PROGRAM prgCS4
VAR
	fbAlfen1					: FB_ECS_Alfen_NG9xx_Platform;						//{#lynus.ag#()}
	fbAlfen2					: FB_ECS_Alfen_NG9xx_Platform;						//{#lynus.ag#()}
	fbAlfen3					: FB_ECS_Alfen_NG9xx_Platform;						//{#lynus.ag#()}
	fbAlfen4					: FB_ECS_Alfen_NG9xx_Platform;						//{#lynus.ag#()}
	fbAlfen5					: FB_ECS_Alfen_NG9xx_Platform;						//{#lynus.ag#()}
	fbAlfen6					: FB_ECS_Alfen_NG9xx_Platform;						//{#lynus.ag#()}
	fbAlfen7					: FB_ECS_Alfen_NG9xx_Platform;						//{#lynus.ag#()}
	fbAlfen8					: FB_ECS_Alfen_NG9xx_Platform;						//{#lynus.ag#()}
	fbAlfen9					: FB_ECS_Alfen_NG9xx_Platform;						//{#lynus.ag#()}
	fbAlfen10					: FB_ECS_Alfen_NG9xx_Platform;						//{#lynus.ag#()}
	
	byErrorWarningUV1_1			: BYTE;												//{#lynus.ag#()}
	rChargingTimeInMinUV1_1		: REAL;												//{#lynus.ag#()}
	lrPowerUV1_1				: LREAL;											//{#lynus.ag#()}
	wStateUV1_1					: WORD;												//{#lynus.ag#()}
	lrEnergySessionUV1_1		: LREAL;											//{#lynus.ag#()}
	lrTotalEnergyUV1_1			: LREAL;											//{#lynus.ag#()}
	
	byErrorWarningUV1_2			: BYTE;												//{#lynus.ag#()}
	rChargingTimeInMinUV1_2		: REAL;												//{#lynus.ag#()}
	lrPowerUV1_2				: LREAL;											//{#lynus.ag#()}
	wStateUV1_2					: WORD;												//{#lynus.ag#()}
	lrEnergySessionUV1_2		: LREAL;											//{#lynus.ag#()}
	lrTotalEnergyUV1_2			: LREAL;											//{#lynus.ag#()}
	
	byErrorWarningUV1_3			: BYTE;												//{#lynus.ag#()}
	rChargingTimeInMinUV1_3		: REAL;												//{#lynus.ag#()}
	lrPowerUV1_3				: LREAL;											//{#lynus.ag#()}
	wStateUV1_3					: WORD;												//{#lynus.ag#()}
	lrEnergySessionUV1_3		: LREAL;											//{#lynus.ag#()}
	lrTotalEnergyUV1_3			: LREAL;											//{#lynus.ag#()}
	
	byErrorWarningUV1_4			: BYTE;												//{#lynus.ag#()}
	rChargingTimeInMinUV1_4		: REAL;												//{#lynus.ag#()}
	lrPowerUV1_4				: LREAL;											//{#lynus.ag#()}
	wStateUV1_4					: WORD;												//{#lynus.ag#()}
	lrEnergySessionUV1_4		: LREAL;											//{#lynus.ag#()}
	lrTotalEnergyUV1_4			: LREAL;											//{#lynus.ag#()}
	
	byErrorWarningUV1_5			: BYTE;												//{#lynus.ag#()}
	rChargingTimeInMinUV1_5		: REAL;												//{#lynus.ag#()}
	lrPowerUV1_5				: LREAL;											//{#lynus.ag#()}
	wStateUV1_5					: WORD;												//{#lynus.ag#()}
	lrEnergySessionUV1_5		: LREAL;											//{#lynus.ag#()}
	lrTotalEnergyUV1_5			: LREAL;											//{#lynus.ag#()}
	
	byErrorWarningUV1_6			: BYTE;												//{#lynus.ag#()}
	rChargingTimeInMinUV1_6		: REAL;												//{#lynus.ag#()}
	lrPowerUV1_6				: LREAL;											//{#lynus.ag#()}
	wStateUV1_6					: WORD;												//{#lynus.ag#()}
	lrEnergySessionUV1_6		: LREAL;											//{#lynus.ag#()}
	lrTotalEnergyUV1_6			: LREAL;											//{#lynus.ag#()}
	
	byErrorWarningUV1_7			: BYTE;												//{#lynus.ag#()}
	rChargingTimeInMinUV1_7		: REAL;												//{#lynus.ag#()}
	lrPowerUV1_7				: LREAL;											//{#lynus.ag#()}
	wStateUV1_7					: WORD;												//{#lynus.ag#()}
	lrEnergySessionUV1_7		: LREAL;											//{#lynus.ag#()}
	lrTotalEnergyUV1_7			: LREAL;											//{#lynus.ag#()}
	
	byErrorWarningUV1_8			: BYTE;												//{#lynus.ag#()}
	rChargingTimeInMinUV1_8		: REAL;												//{#lynus.ag#()}
	lrPowerUV1_8				: LREAL;											//{#lynus.ag#()}
	wStateUV1_8					: WORD;												//{#lynus.ag#()}
	lrEnergySessionUV1_8		: LREAL;											//{#lynus.ag#()}
	lrTotalEnergyUV1_8			: LREAL;											//{#lynus.ag#()}
	
	byErrorWarningUV1_9			: BYTE;												//{#lynus.ag#()}
	rChargingTimeInMinUV1_9		: REAL;												//{#lynus.ag#()}
	lrPowerUV1_9				: LREAL;											//{#lynus.ag#()}
	wStateUV1_9					: WORD;												//{#lynus.ag#()}
	lrEnergySessionUV1_9		: LREAL;											//{#lynus.ag#()}
	lrTotalEnergyUV1_9			: LREAL;											//{#lynus.ag#()}
	
	byErrorWarningUV1_10		: BYTE;												//{#lynus.ag#()}
	rChargingTimeInMinUV1_10	: REAL;												//{#lynus.ag#()}
	lrPowerUV1_10				: LREAL;											//{#lynus.ag#()}
	wStateUV1_10				: WORD;												//{#lynus.ag#()}
	lrEnergySessionUV1_10		: LREAL;											//{#lynus.ag#()}
	lrTotalEnergyUV1_10			: LREAL;											//{#lynus.ag#()}
END_VAR

(*---------------------------------------------CS1-----------------------------------------------------------*)

fbAlfen1(
	bEnable:= , 
	bPowerDataInvers:= , 
	byElectricFuseLine:= 3, 
	byUnitID_Socket1:= 1, 
	byUnitID_Socket2:= , 
	byNumberOfSockets:= 1, 
	byNumberOfConnectionWire:= 1, 
	diNrOfEMS_IN:= prgEMS.fbEMS2.diNrOfEMS_OUT, 
	diNrOfEM_IN_CS:= , 
	sIPAdress:= '192.168.1.41', 
	stSetupECS:= , 
	stDataECS=> , 
	diNrOfECS_OUT=> );

		byErrorWarningUV1_1 := fbAlfen1.stDataECS.byErrorWarning;	
			rChargingTimeInMinUV1_1 := fbAlfen1.stDataECS.arrChargingTimeInMin[1];
				lrPowerUV1_1 := fbAlfen1.stDataECS.lrTotalPower;	
					wStateUV1_1 := fbAlfen1.stDataECS.arrSocketStateECS[1];
						lrEnergySessionUV1_1 := fbAlfen1.stDataECS.arrSocketEnergySession[1];
							lrTotalEnergyUV1_1 := fbAlfen1.stDataECS.lrTotalCounterEnergy_Consumption;	
	
(*---------------------------------------------CS2-----------------------------------------------------------*)
	
fbAlfen2(
	bEnable:= , 
	bPowerDataInvers:= , 
	byElectricFuseLine:= 3, 
	byUnitID_Socket1:= 1, 
	byUnitID_Socket2:= , 
	byNumberOfSockets:= 1, 
	byNumberOfConnectionWire:= 1, 
	diNrOfEMS_IN:= prgEMS.fbEMS2.diNrOfEMS_OUT, 
	diNrOfEM_IN_CS:= , 
	sIPAdress:= '192.168.1.42', 
	stSetupECS:= , 
	stDataECS=> , 
	diNrOfECS_OUT=> );

		byErrorWarningUV1_2 := fbAlfen2.stDataECS.byErrorWarning;
			rChargingTimeInMinUV1_2 := fbAlfen2.stDataECS.arrChargingTimeInMin[1];;
				lrPowerUV1_2 := fbAlfen2.stDataECS.lrTotalPower;	
					wStateUV1_2 := fbAlfen2.stDataECS.arrSocketStateECS[1];
						lrEnergySessionUV1_2 := fbAlfen2.stDataECS.arrSocketEnergySession[1];
							lrTotalEnergyUV1_2 := fbAlfen2.stDataECS.lrTotalCounterEnergy_Consumption;
	
(*---------------------------------------------CS3-----------------------------------------------------------*)	

fbAlfen3(
	bEnable:= , 
	bPowerDataInvers:= , 
	byElectricFuseLine:= 3, 
	byUnitID_Socket1:= 1, 
	byUnitID_Socket2:= , 
	byNumberOfSockets:= 1, 
	byNumberOfConnectionWire:= 1, 
	diNrOfEMS_IN:= prgEMS.fbEMS2.diNrOfEMS_OUT, 
	diNrOfEM_IN_CS:= , 
	sIPAdress:= '192.168.1.43', 
	stSetupECS:= , 
	stDataECS=> , 
	diNrOfECS_OUT=> );

		byErrorWarningUV1_3 := fbAlfen3.stDataECS.byErrorWarning;
			rChargingTimeInMinUV1_3 := fbAlfen3.stDataECS.arrChargingTimeInMin[1];	
				lrPowerUV1_3 := fbAlfen3.stDataECS.lrTotalPower;	
					wStateUV1_3 := fbAlfen3.stDataECS.arrSocketStateECS[1];
						lrEnergySessionUV1_3 := fbAlfen3.stDataECS.arrSocketEnergySession[1];
							lrTotalEnergyUV1_3 := fbAlfen3.stDataECS.lrTotalCounterEnergy_Consumption;	
	
(*---------------------------------------------CS4-----------------------------------------------------------*)	

fbAlfen4(
	bEnable:= , 
	bPowerDataInvers:= , 
	byElectricFuseLine:= 3, 
	byUnitID_Socket1:= 1, 
	byUnitID_Socket2:= , 
	byNumberOfSockets:= 1, 
	byNumberOfConnectionWire:= 1, 
	diNrOfEMS_IN:= prgEMS.fbEMS2.diNrOfEMS_OUT, 
	diNrOfEM_IN_CS:= , 
	sIPAdress:= '192.168.1.44', 
	stSetupECS:= , 
	stDataECS=> , 
	diNrOfECS_OUT=> );

		byErrorWarningUV1_4 := fbAlfen4.stDataECS.byErrorWarning;
			rChargingTimeInMinUV1_4 := fbAlfen4.stDataECS.arrChargingTimeInMin[1];
				lrPowerUV1_4 := fbAlfen4.stDataECS.lrTotalPower;	
					wStateUV1_4 := fbAlfen4.stDataECS.arrSocketStateECS[1];
						lrEnergySessionUV1_4 := fbAlfen4.stDataECS.arrSocketEnergySession[1];
							lrTotalEnergyUV1_4 := fbAlfen4.stDataECS.lrTotalCounterEnergy_Consumption;
	
(*---------------------------------------------CS5-----------------------------------------------------------*)	

fbAlfen5(
	bEnable:= , 
	bPowerDataInvers:= , 
	byElectricFuseLine:= 3, 
	byUnitID_Socket1:= 1, 
	byUnitID_Socket2:= , 
	byNumberOfSockets:= 1, 
	byNumberOfConnectionWire:= 1, 
	diNrOfEMS_IN:= prgEMS.fbEMS2.diNrOfEMS_OUT, 
	diNrOfEM_IN_CS:= , 
	sIPAdress:= '192.168.1.45', 
	stSetupECS:= , 
	stDataECS=> , 
	diNrOfECS_OUT=> );

		byErrorWarningUV1_5 := fbAlfen5.stDataECS.byErrorWarning;
			rChargingTimeInMinUV1_5 := fbAlfen5.stDataECS.arrChargingTimeInMin[1];
				lrPowerUV1_5 := fbAlfen5.stDataECS.lrTotalPower;	
					wStateUV1_5 := fbAlfen5.stDataECS.arrSocketStateECS[1];
						lrEnergySessionUV1_5 := fbAlfen5.stDataECS.arrSocketEnergySession[1];
							lrTotalEnergyUV1_5 := fbAlfen5.stDataECS.lrTotalCounterEnergy_Consumption;	
	
(*---------------------------------------------CS6-----------------------------------------------------------*)	

fbAlfen6(
	bEnable:= , 
	bPowerDataInvers:= , 
	byElectricFuseLine:= 3, 
	byUnitID_Socket1:= 1, 
	byUnitID_Socket2:= , 
	byNumberOfSockets:= 1, 
	byNumberOfConnectionWire:= 1, 
	diNrOfEMS_IN:= prgEMS.fbEMS2.diNrOfEMS_OUT, 
	diNrOfEM_IN_CS:= , 
	sIPAdress:= '192.168.1.46', 
	stSetupECS:= , 
	stDataECS=> , 
	diNrOfECS_OUT=> );

		byErrorWarningUV1_6 := fbAlfen6.stDataECS.byErrorWarning;
			rChargingTimeInMinUV1_6 := fbAlfen6.stDataECS.arrChargingTimeInMin[1];
				lrPowerUV1_6 := fbAlfen6.stDataECS.lrTotalPower;	
					wStateUV1_6 := fbAlfen6.stDataECS.arrSocketStateECS[1];
						lrEnergySessionUV1_6 := fbAlfen6.stDataECS.arrSocketEnergySession[1];
							lrTotalEnergyUV1_6 := fbAlfen6.stDataECS.lrTotalCounterEnergy_Consumption;
	
(*---------------------------------------------CS7-----------------------------------------------------------*)	

fbAlfen7(
	bEnable:= , 
	bPowerDataInvers:= , 
	byElectricFuseLine:= 3, 
	byUnitID_Socket1:= 1, 
	byUnitID_Socket2:= , 
	byNumberOfSockets:= 1, 
	byNumberOfConnectionWire:= 1, 
	diNrOfEMS_IN:= prgEMS.fbEMS2.diNrOfEMS_OUT, 
	diNrOfEM_IN_CS:= , 
	sIPAdress:= '192.168.1.47', 
	stSetupECS:= , 
	stDataECS=> , 
	diNrOfECS_OUT=> );

		byErrorWarningUV1_7 := fbAlfen7.stDataECS.byErrorWarning;
			rChargingTimeInMinUV1_7 := fbAlfen7.stDataECS.arrChargingTimeInMin[1];
				lrPowerUV1_7 := fbAlfen7.stDataECS.lrTotalPower;	
					wStateUV1_7 := fbAlfen7.stDataECS.arrSocketStateECS[1];
						lrEnergySessionUV1_7 := fbAlfen7.stDataECS.arrSocketEnergySession[1];
							lrTotalEnergyUV1_7 := fbAlfen7.stDataECS.lrTotalCounterEnergy_Consumption;
	
(*---------------------------------------------CS8-----------------------------------------------------------*)	

fbAlfen8(
	bEnable:= , 
	bPowerDataInvers:= , 
	byElectricFuseLine:= 3, 
	byUnitID_Socket1:= 1, 
	byUnitID_Socket2:= , 
	byNumberOfSockets:= 1, 
	byNumberOfConnectionWire:= 1, 
	diNrOfEMS_IN:= prgEMS.fbEMS2.diNrOfEMS_OUT, 
	diNrOfEM_IN_CS:= , 
	sIPAdress:= '192.168.1.48', 
	stSetupECS:= , 
	stDataECS=> , 
	diNrOfECS_OUT=> );

		byErrorWarningUV1_8 := fbAlfen8.stDataECS.byErrorWarning;
			rChargingTimeInMinUV1_8 := fbAlfen8.stDataECS.arrChargingTimeInMin[1];
				lrPowerUV1_8 := fbAlfen8.stDataECS.lrTotalPower;	
					wStateUV1_8 := fbAlfen8.stDataECS.arrSocketStateECS[1];
						lrEnergySessionUV1_8 := fbAlfen8.stDataECS.arrSocketEnergySession[1];
							lrTotalEnergyUV1_8 := fbAlfen8.stDataECS.lrTotalCounterEnergy_Consumption;
	
(*---------------------------------------------CS9-----------------------------------------------------------*)	

fbAlfen9(
	bEnable:= , 
	bPowerDataInvers:= , 
	byElectricFuseLine:= 4, 
	byUnitID_Socket1:= 1, 
	byUnitID_Socket2:= , 
	byNumberOfSockets:= 1, 
	byNumberOfConnectionWire:= 1, 
	diNrOfEMS_IN:= prgEMS.fbEMS2.diNrOfEMS_OUT, 
	diNrOfEM_IN_CS:= , 
	sIPAdress:= '192.168.1.49', 
	stSetupECS:= , 
	stDataECS=> , 
	diNrOfECS_OUT=> );

		byErrorWarningUV1_9 := fbAlfen9.stDataECS.byErrorWarning;	
			rChargingTimeInMinUV1_9 := fbAlfen9.stDataECS.arrChargingTimeInMin[1];
				lrPowerUV1_9 := fbAlfen9.stDataECS.lrTotalPower;	
					wStateUV1_9 := fbAlfen9.stDataECS.arrSocketStateECS[1];
						lrEnergySessionUV1_9 := fbAlfen9.stDataECS.arrSocketEnergySession[1];
							lrTotalEnergyUV1_9 := fbAlfen9.stDataECS.lrTotalCounterEnergy_Consumption;
	
(*---------------------------------------------CS10-----------------------------------------------------------*)	

fbAlfen10(
	bEnable:= , 
	bPowerDataInvers:= , 
	byElectricFuseLine:= 4, 
	byUnitID_Socket1:= 1, 
	byUnitID_Socket2:= , 
	byNumberOfSockets:= 1, 
	byNumberOfConnectionWire:= 1, 
	diNrOfEMS_IN:= prgEMS.fbEMS2.diNrOfEMS_OUT, 
	diNrOfEM_IN_CS:= , 
	sIPAdress:= '192.168.1.50', 
	stSetupECS:= , 
	stDataECS=> , 
	diNrOfECS_OUT=> );

		byErrorWarningUV1_10 := fbAlfen10.stDataECS.byErrorWarning;	
			rChargingTimeInMinUV1_10 := fbAlfen10.stDataECS.arrChargingTimeInMin[1];
				lrPowerUV1_10 := fbAlfen10.stDataECS.lrTotalPower;	
					wStateUV1_10 := fbAlfen10.stDataECS.arrSocketStateECS[1];
						lrEnergySessionUV1_10 := fbAlfen10.stDataECS.arrSocketEnergySession[1];
							lrTotalEnergyUV1_10 := fbAlfen10.stDataECS.lrTotalCounterEnergy_Consumption;

END_PROGRAM

(* stored: Version 1.1.0.1, ProductVersion 3.1.4024.9
   POU prgCS4: Id {23a22fdd-e742-43ff-9be5-ffc516565f3b}, SpecialFunc None *)
